(* PLC project Unnamed, Unknown Unnamed 1 *)
(* stored: creationDateTime 2026-04-01T18:01:00, modificationDateTime 2026-04-01T18:01:00 *)

PROGRAM main
  VAR
    BTN_ON_1 AT %IX0.3 : BOOL;
    BTN_ON_2 AT %IX0.5 : BOOL;
    OUT_1 AT %QX0.0 : BOOL;
    OUT_2 AT %QX0.1 : BOOL;
    BTN_OFF_1 AT %IX0.4 : BOOL;
    BTN_OFF_2 AT %IX0.6 : BOOL;
  END_VAR
  VAR
    OUT_3 : BOOL;
  END_VAR
  VAR  (* added by the conversion: wires and edge detectors of the diagram *)
    R_TRIG1 : R_TRIG;
    R_TRIG2 : R_TRIG;
  END_VAR

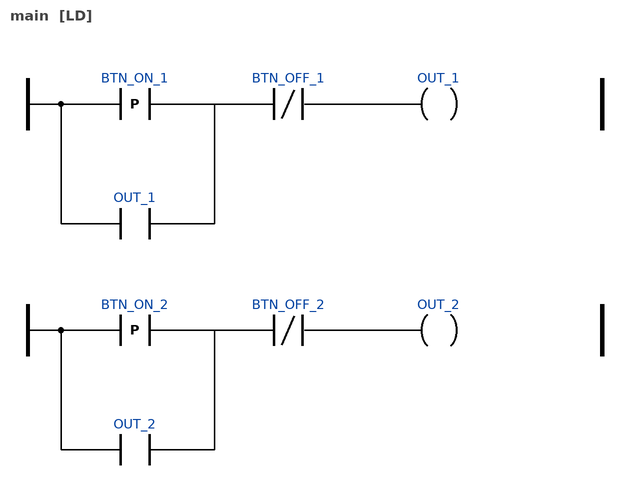
(* LD diagram, written out as Structured Text *)
R_TRIG1(CLK := BTN_ON_1);
OUT_1 := (R_TRIG1.Q OR OUT_1) AND NOT BTN_OFF_1;
R_TRIG2(CLK := BTN_ON_2);
OUT_2 := (R_TRIG2.Q OR OUT_2) AND NOT BTN_OFF_2;
END_PROGRAM

CONFIGURATION Config0
  RESOURCE Res0 ON PLC
    TASK task0(INTERVAL := T#20ms, PRIORITY := 1);
    PROGRAM instance0 WITH task0 : main;
  END_RESOURCE
END_CONFIGURATION
